INTERFACE I_HaveMetadata EXTENDS __SYSTEM.IQueryInterface

METHOD AddMetadatum
VAR_INPUT
	Metadatum : I_Metadatum;
END_VAR
END_METHOD

METHOD PUBLIC GetMetadata : I_Metadata
VAR_INPUT
END_VAR
END_METHOD

METHOD PUBLIC TryGetMetadatumByName : BOOL
VAR_INPUT
	Name : T_MAXSTRING;
	Destination : REFERENCE TO I_Metadatum;
END_VAR
END_METHOD

END_INTERFACE

(* stored: Version 1.1.0.1, ProductVersion 3.1.4024.12
   Itf I_HaveMetadata: Id {96f646d1-a4c9-0134-213d-25e203a1beca}
   Method AddMetadatum: Id {c58c1d1e-b1d1-0e7a-041f-b8740747188f}
   Method GetMetadata: Id {509044e7-6ece-0a78-0078-53d3ca44d828}
   Method TryGetMetadatumByName: Id {8bd144a5-6123-06fd-0e73-e7fee3e3c69c} *)
